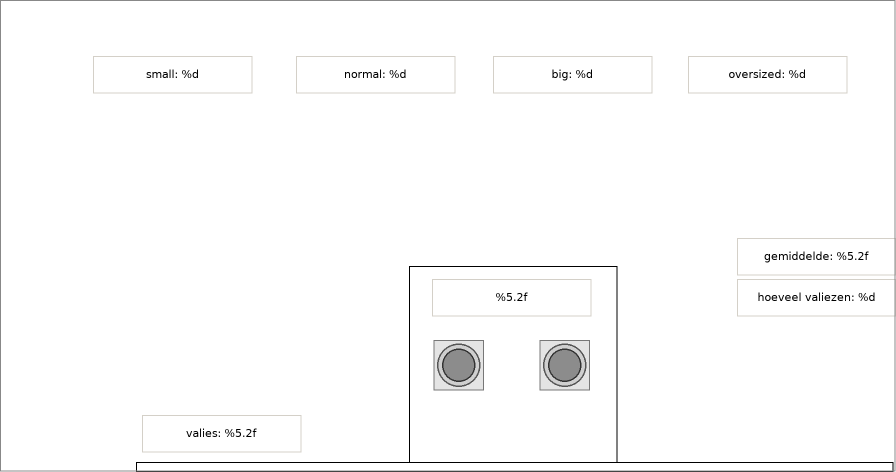
VISUALIZATION Visualization  // 896x472
    Rectangle (409,266 208x206)
    PushSwitch (432,340 53x50), variable: analogSignals_ex07.OK.DI_Input, behaviour: TOGGLE, style: Switch-PushSwitch-Gray
    PushSwitch (538,340 53x50), variable: analogSignals_ex07.Reset.DI_Input, behaviour: TOGGLE, style: Switch-PushSwitch-Gray
    Rectangle (136,462 757x10)
    Textfield (432,279 159x37), "%5.2f", text variable: analogSignals_ex07.weight
    Textfield (93,56 159x37), "small: %d", text variable: analogSignals_ex07.tellersmall.CV
    Textfield (296,56 159x37), "normal: %d", text variable: analogSignals_ex07.tellernormal.CV
    Textfield (493,56 159x37), "big: %d", text variable: analogSignals_ex07.tellerbig.CV
    Textfield (688,56 159x37), "oversized: %d", text variable: analogSignals_ex07.telleroversized.CV
    Textfield (737,238 159x37), "gemiddelde: %5.2f", text variable: analogSignals_ex07.gemiddelde4.fAverage
    Textfield (737,279 159x37), "hoeveel valiezen: %d", text variable: analogSignals_ex07.gemiddelde4.nCount
    Textfield (142,415 159x37), "valies: %5.2f", text variable: analogSignals_ex07.weightsensor
        OnMouseClick: write the text variable via VisuDialogs.Numpad, min 4, max 20
END_VISUALIZATION

(* stored: Version 1.1.0.1
   Visu Visualization: Id {85a4990d-d78f-4ca6-b6c3-26895e3a52ec} *)
